PROGRAM _Home


VAR


    END_VAR

END_PROGRAM

END_PROGRAM

CASE HomeStep OF


0:

bLimitHomeZ := TRUE;

IF mcStepLimitSwitchZ.Done THEN

bLimitHomeZ := FALSE;

HomeStep := HomeStep + 1;

            END_IF


1:

bPulseHomeZ := TRUE;

IF mcStepReferenceZ.done THEN

bPulseHomeZ := FALSE;

HomeStep := HomeStep + 1;

            END_IF


2:
            bFinishHomeZ := TRUE;

IF mcFinishHomingZ.done THEN

bFinishHomeZ := FALSE;

HomeStep := HomeStep + 1;

            END_IF



3:
            bLimitHomeX := TRUE;

bLimitHomeY := TRUE;

IF mcStepLimitSwitchX.done AND mcStepLimitSwitchY.done THEN

bLimitHomeX := FALSE;

bLimitHomeY := FALSE;

HomeStep := HomeStep + 1;

            END_IF


4:
            bPulseHomeX := TRUE;

bPulseHomeY := TRUE;

IF mcStepReferenceX.Done AND mcStepReferenceY.Done THEN

bPulseHomeX := FALSE;

bPulseHomeY := FALSE;

HomeStep := HomeStep + 1;

            END_IF


5:
            bFinishHomeX := TRUE;

bFinishHomeY := TRUE;

IF mcFinishHomingX.Done AND mcFinishHomingY.Done THEN

bFinishHomeX := FALSE;

bFinishHomeY := FALSE;

HomeStep := HomeStep + 1;

            END_IF


6:

bOffsetHomeX := TRUE;

bOffsetHomeY := TRUE;

bOffsetHomeZ := TRUE;

IF mcSetOffsetHomePosX.Done
 AND mcSetOffsetHomePosY.Done
 AND mcSetOffsetHomePosZ.Done THEN

bOffsetHomeX := FALSE;

bOffsetHomeY := FALSE;

bOffsetHomeZ := FALSE;

homedone := TRUE;

            END_IF

    END_CASE

ACTION _StepLimitSwitch:
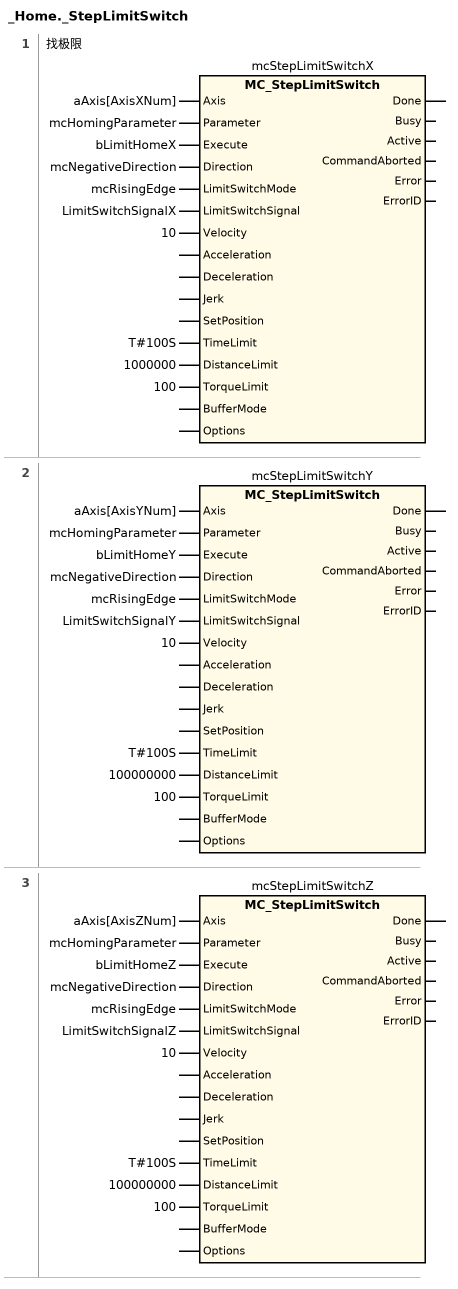
// NETWORK 1: 找极限
mcStepLimitSwitchX(
    Axis := aAxis[AxisXNum],
    Parameter := mcHomingParameter,
    Execute := bLimitHomeX,
    Direction := mcNegativeDirection,
    LimitSwitchMode := mcRisingEdge,
    LimitSwitchSignal := LimitSwitchSignalX,
    Velocity := 10,
    TimeLimit := T#100S,
    DistanceLimit := 1000000,
    TorqueLimit := 100); // MC_StepLimitSwitch

// NETWORK 2
mcStepLimitSwitchY(
    Axis := aAxis[AxisYNum],
    Parameter := mcHomingParameter,
    Execute := bLimitHomeY,
    Direction := mcNegativeDirection,
    LimitSwitchMode := mcRisingEdge,
    LimitSwitchSignal := LimitSwitchSignalY,
    Velocity := 10,
    TimeLimit := T#100S,
    DistanceLimit := 100000000,
    TorqueLimit := 100); // MC_StepLimitSwitch

// NETWORK 3
mcStepLimitSwitchZ(
    Axis := aAxis[AxisZNum],
    Parameter := mcHomingParameter,
    Execute := bLimitHomeZ,
    Direction := mcNegativeDirection,
    LimitSwitchMode := mcRisingEdge,
    LimitSwitchSignal := LimitSwitchSignalZ,
    Velocity := 10,
    TimeLimit := T#100S,
    DistanceLimit := 100000000,
    TorqueLimit := 100); // MC_StepLimitSwitch

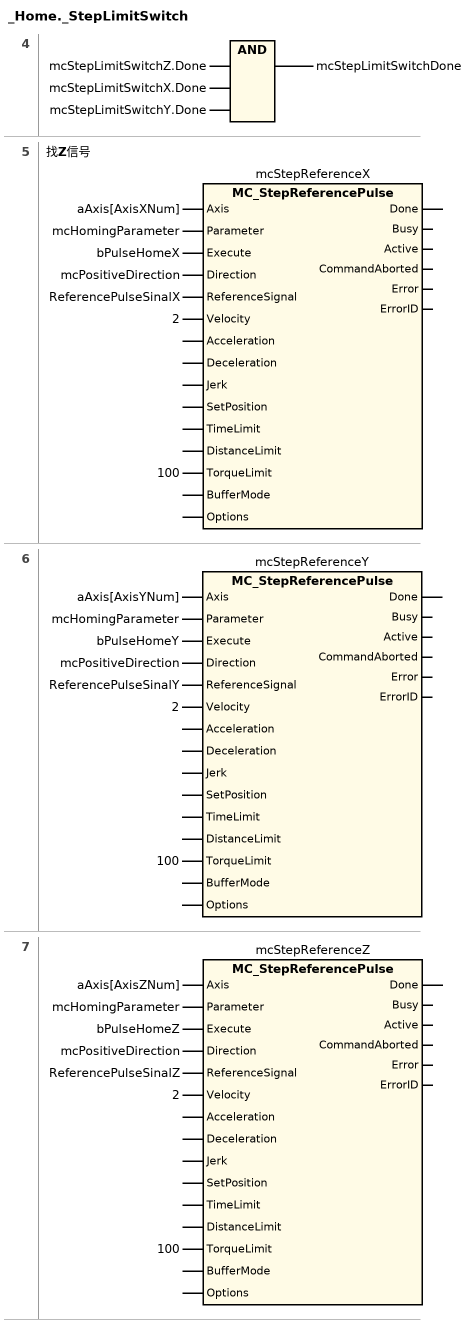
// NETWORK 4
mcStepLimitSwitchDone := mcStepLimitSwitchZ.Done AND mcStepLimitSwitchX.Done AND mcStepLimitSwitchY.Done;

// NETWORK 5: 找Z信号
mcStepReferenceX(
    Axis := aAxis[AxisXNum],
    Parameter := mcHomingParameter,
    Execute := bPulseHomeX,
    Direction := mcPositiveDirection,
    ReferenceSignal := ReferencePulseSinalX,
    Velocity := 2,
    TorqueLimit := 100); // MC_StepReferencePulse

// NETWORK 6
mcStepReferenceY(
    Axis := aAxis[AxisYNum],
    Parameter := mcHomingParameter,
    Execute := bPulseHomeY,
    Direction := mcPositiveDirection,
    ReferenceSignal := ReferencePulseSinalY,
    Velocity := 2,
    TorqueLimit := 100); // MC_StepReferencePulse

// NETWORK 7
mcStepReferenceZ(
    Axis := aAxis[AxisZNum],
    Parameter := mcHomingParameter,
    Execute := bPulseHomeZ,
    Direction := mcPositiveDirection,
    ReferenceSignal := ReferencePulseSinalZ,
    Velocity := 2,
    TorqueLimit := 100); // MC_StepReferencePulse

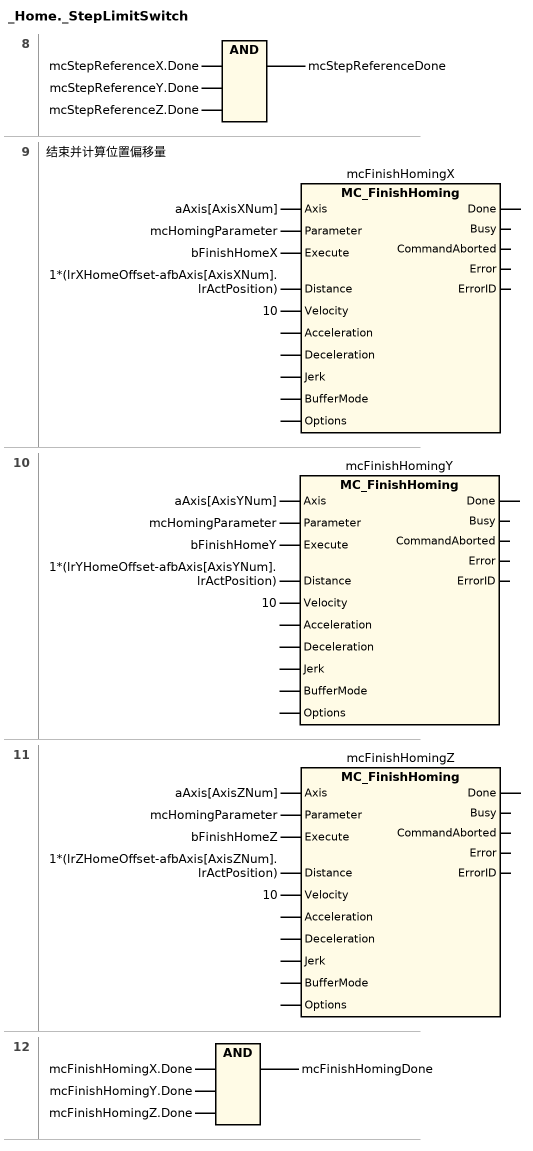
// NETWORK 8
mcStepReferenceDone := mcStepReferenceX.Done AND mcStepReferenceY.Done AND mcStepReferenceZ.Done;

// NETWORK 9: 结束并计算位置偏移量
mcFinishHomingX(
    Axis := aAxis[AxisXNum],
    Parameter := mcHomingParameter,
    Execute := bFinishHomeX,
    Distance := 1*(lrXHomeOffset-afbAxis[AxisXNum].lrActPosition),
    Velocity := 10); // MC_FinishHoming

// NETWORK 10
mcFinishHomingY(
    Axis := aAxis[AxisYNum],
    Parameter := mcHomingParameter,
    Execute := bFinishHomeY,
    Distance := 1*(lrYHomeOffset-afbAxis[AxisYNum].lrActPosition),
    Velocity := 10); // MC_FinishHoming

// NETWORK 11
mcFinishHomingZ(
    Axis := aAxis[AxisZNum],
    Parameter := mcHomingParameter,
    Execute := bFinishHomeZ,
    Distance := 1*(lrZHomeOffset-afbAxis[AxisZNum].lrActPosition),
    Velocity := 10); // MC_FinishHoming

// NETWORK 12
mcFinishHomingDone := mcFinishHomingX.Done AND mcFinishHomingY.Done AND mcFinishHomingZ.Done;

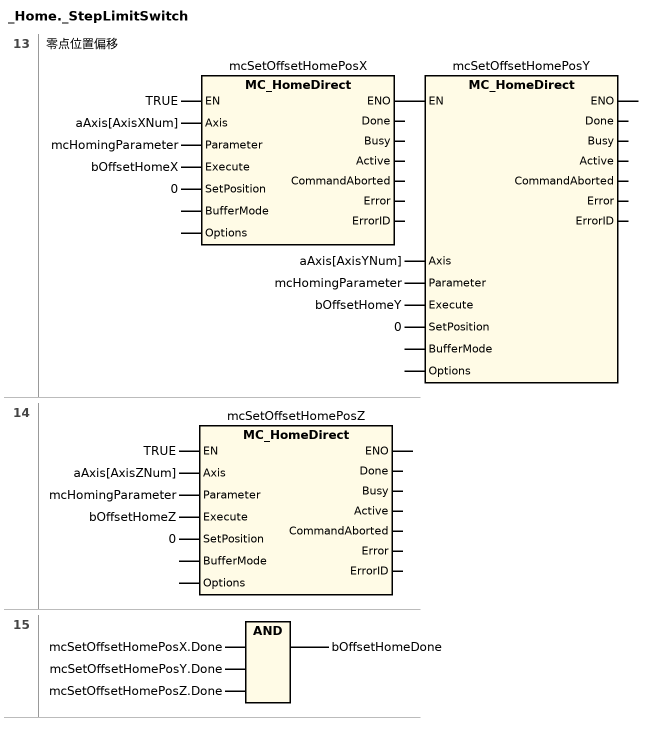
// NETWORK 13: 零点位置偏移
mcSetOffsetHomePosX(
    Axis := aAxis[AxisXNum],
    Parameter := mcHomingParameter,
    Execute := bOffsetHomeX,
    SetPosition := 0); // MC_HomeDirect
mcSetOffsetHomePosY(
    Axis := aAxis[AxisYNum],
    Parameter := mcHomingParameter,
    Execute := bOffsetHomeY,
    SetPosition := 0); // MC_HomeDirect

// NETWORK 14
mcSetOffsetHomePosZ(
    Axis := aAxis[AxisZNum],
    Parameter := mcHomingParameter,
    Execute := bOffsetHomeZ,
    SetPosition := 0); // MC_HomeDirect

// NETWORK 15
bOffsetHomeDone := mcSetOffsetHomePosX.Done AND mcSetOffsetHomePosY.Done AND mcSetOffsetHomePosZ.Done;
END_ACTION

END_PROGRAM

(* stored: Version 1.1.0.1, ProductVersion 3.1.4024.12
   POU _Home: Id {afdb9434-577b-41f5-ad59-27efb8bb840b}, SpecialFunc None
   Action _StepLimitSwitch: Id {73f00320-841c-45ad-b3df-dd42b4f579ad} *)
